(* CoDeSys 2.3 export: FC_MQTT_CLEARTELEGRAM_V10.EXP *)

(* POU _Generic/Mqtt/Intern/FC_Mqtt_ClearTelegram_V10, ST *)
FUNCTION FC_Mqtt_ClearTelegram_V10 : BOOL
VAR_IN_OUT
	stMqttTelegram	: ST_MqttTelegram;
	stMqttSettings	: ST_MqttSettings;
END_VAR
VAR
END_VAR
MEMSET(
	destAddr	:= ADR(stMqttTelegram.arMqttData),
	fillByte  	:= 0,
	n			:= stMqttSettings.iTelegramSize
);

stMqttTelegram.nDataLength := 0;
END_FUNCTION
